% RSLogix 500 project CAR WASHING PROCESS_BAK006.RSS, saved by version 8.30.00.16 %
PROJECT "UNTITLED"    % processor: Bul.1763 MicroLogix 1100 Series B %

PROGRAM FILES
  LAD 2   8 rungs

DATA FILES
  O0 OUTPUT  4 elements
  I1 INPUT  6 elements
  S2 STATUS  66 elements
  B3 BINARY  46 elements
  T4 TIMER  1 elements
  C5 COUNTER  1 elements
  R6 CONTROL  3 elements
  N7 INTEGER  1 elements
  F8 FLOAT  1 elements

LADDER 2
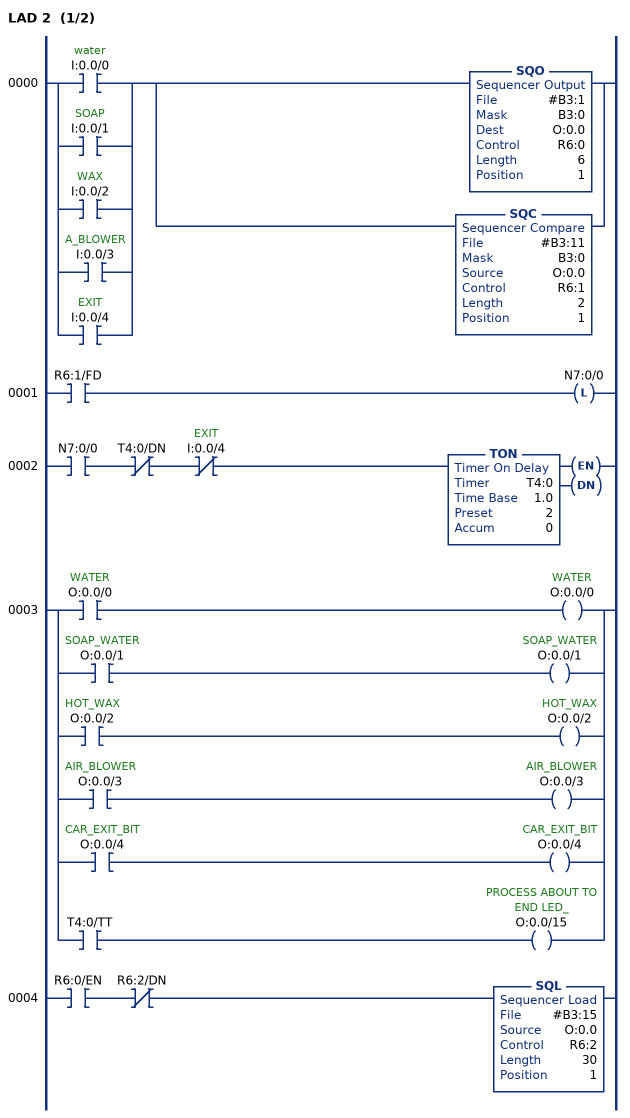
% Rung: 0 %
SOR BST XIC I:0.0/0 NXB XIC I:0.0/1 NXB XIC I:0.0/2 NXB XIC I:0.0/3 NXB XIC I:0.0/4 BND BST SQO #B3:1 B3:0 O:0.0 R6:0 6 1 NXB SQC #B3:11 B3:0 O:0.0 R6:1 2 1 BND EOR
%   I:0.0/0  "water" %
%   I:0.0/1  SOAP %
%   I:0.0/2  "WAX" %
%   I:0.0/3  A_BLOWER %
%   I:0.0/4  "EXIT" %
%   B3:1  SYS %
%   B3:0  MUSK %
% Rung: 1 %
SOR XIC R6:1/FD OTL N7:0/0 EOR
% Rung: 2 %
SOR XIC N7:0/0 XIO T4:0/DN XIO I:0.0/4 TON T4:0 1.0 2 0 EOR
%   I:0.0/4  "EXIT" %
% Rung: 3 %
SOR BST XIC O:0.0/0 OTE O:0.0/0 NXB XIC O:0.0/1 OTE O:0.0/1 NXB XIC O:0.0/2 OTE O:0.0/2 NXB XIC O:0.0/3 OTE O:0.0/3 NXB XIC O:0.0/4 OTE O:0.0/4 NXB XIC T4:0/TT OTE O:0.0/15 BND EOR
%   O:0.0/0  WATER %
%   O:0.0/1  SOAP_WATER %
%   O:0.0/2  HOT_WAX %
%   O:0.0/3  AIR_BLOWER %
%   O:0.0/4  CAR_EXIT_BIT %
%   O:0.0/15  LED_  "PROCESS ABOUT TO END" %
% Rung: 4 %
SOR XIC R6:0/EN XIO R6:2/DN SQL #B3:15 O:0.0 R6:2 30 1 EOR

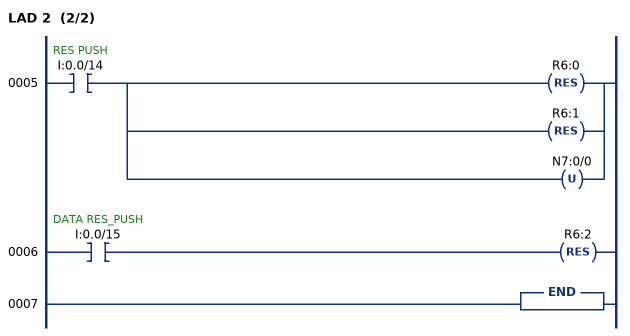
% Rung: 5 %
SOR XIC I:0.0/14 BST RES R6:0 NXB RES R6:1 NXB OTU N7:0/0 BND EOR
%   I:0.0/14  "RES PUSH" %
% Rung: 6 %
SOR XIC I:0.0/15 RES R6:2 EOR
%   I:0.0/15  RES_PUSH  "DATA" %
% Rung: 7 %
SOR END EOR

DATA TABLE (non-zero values as saved)
DATA B3
% B3:0 % 0X0FFF 0X0000 0X0001 0X0003 0X0001 0X0004 0X0008 0X0010 0X0000 0X0000
% B3:10 % 0X0000 0X0008 0X0008 0X0000 0X0000 0X0000 0X0001 0X0003 0X0001 0X0004
% B3:20 % 0X8008 0X8010 0X0001 0X0003 0X0001 0X0004 0X0008 0X0010 0X0001 0X0003
% B3:30 % 0X0001 0X0004 0X0008 0X0010 0X8001 0X0000 0X0000 0X0000 0X0000 0X0000
DATA T4
% .PRE .ACC %
% T4:0 % 2 0
DATA R6
% .LEN .POS %
% R6:0 % 6 1
% R6:1 % 2 1
% R6:2 % 30 1
